FUNCTION_BLOCK Crane_MoveToStack EXTENDS Crane_MoveBase
VAR_INPUT
END_VAR
VAR_OUTPUT
END_VAR
VAR
	m_precondition: ComparisonExpression(EProcessVariables.Crane_CylinderRetracted, EComparisonType.equals, EDataType.binary, TRUE, 0, '', TRUE);
	
	// EProcessVariables.Crane_AtStack = TRUE
	m_postcondition: ComparisonExpression(EProcessVariables.Crane_AtStack, EComparisonType.equals, EDataType.binary, TRUE, 0, '', TRUE);
END_VAR

SUPER^();

PROPERTY AtTarget : BOOL
GET
AtTarget := m_ptrCrane^.AtStack;
END_GET
END_PROPERTY

METHOD FB_init : BOOL
VAR_INPUT
	bInitRetains : BOOL; // if TRUE, the retain variables are initialized (warm start / cold start)
	bInCopyCode : BOOL;  // if TRUE, the instance afterwards gets moved into the copy code (online change)
		
	i_ptrCrane: POINTER TO Crane;
END_VAR
m_ptrCrane := i_ptrCrane;

m_id := EPrimitives.Crane_MoveToStack;
m_timeout := T#30S;

Precondition := m_precondition;
Postcondition := m_postcondition;
END_METHOD

PROPERTY TargetAngle : UINT
GET
TargetAngle := 0;
END_GET
END_PROPERTY

END_FUNCTION_BLOCK

(* stored: Version 1.1.0.1
   POU Crane_MoveToStack: Id {695e069d-1259-46e4-8622-a00bc39a4090}, SpecialFunc None
   Property AtTarget: Id {9298988e-8013-4356-96a0-a81cbf89c627}
   Get Get: Id {9082eeee-cdc1-4e3e-bd1a-e9e7d6542603}
   Method FB_init: Id {4bee316d-c943-4419-919f-e1ed72d8e24c}
   Property TargetAngle: Id {04e90976-00ce-41ef-9fd6-e908437e1290}
   Get Get: Id {3b0eaaa1-57ad-4b97-bd8f-e37c919b51b8} *)
